// TIA Portal V20 export
DATA_BLOCK "GDB_AxisCtrl"   // DB101
{ S7_Optimized_Access := 'TRUE' }
// stored: AutoNumber false, MemoryReserve 0
   VAR
      TOCtrl { S7_SetPoint := 'True'} : Array[1..10] of "UDT_typePosCtrl";
      LKinCtrl { S7_SetPoint := 'True'} : "UDT_typeKinCtrl";
      Measureinput { S7_SetPoint := 'True'} : Array[1..2] of "UDT_typeMeasureInput";
   END_VAR
BEGIN
   LKinCtrl.input.configuration.jogframe.dynamics.path.velocity := 200.0;
   LKinCtrl.input.configuration.jogframe.dynamics.path.acceleration := 2000.0;
   LKinCtrl.input.configuration.jogframe.dynamics.path.deceleration := 2000.0;
   LKinCtrl.input.configuration.jogframe.dynamics.path.jerk := 20000.0;
   LKinCtrl.input.configuration.jogframe.dynamics.orientation.velocity := 50.0;
   LKinCtrl.input.configuration.jogframe.dynamics.orientation.acceleration := 500.0;
   LKinCtrl.input.configuration.jogframe.dynamics.orientation.deceleration := 500.0;
   LKinCtrl.input.configuration.jogframe.dynamics.orientation.jerk := 5000.0;
END_DATA_BLOCK
